// Alias for __SYSTEM.VAR_INFO.
// [use] Stores variable information.
TYPE T_VarInfo : __SYSTEM.VAR_INFO; END_TYPE

(* stored: Version 1.1.0.1
   DUT T_VarInfo: Id {7ad3f699-14d5-080d-2a66-bd491f8a61d3} *)
